//Check if the symbol string is an array, i.e. contains "[ ]"
FUNCTION F_CheckIsArraySymbol : BOOL
VAR_INPUT
    sSymbolName : STRING;
END_VAR
VAR
    iOpenBrackLocation : INT;
    iClosedBracketLocation : INT;
END_VAR

iOpenBrackLocation := FIND(sSymbolName, '[');
iClosedBracketLocation := FIND(sSymbolName, ']');

IF iOpenBrackLocation <> 0 AND iClosedBracketLocation > iOpenBrackLocation THEN
    F_CheckIsArraySymbol := TRUE;

ELSE
    F_CheckIsArraySymbol := FALSE;
END_IF

END_FUNCTION

(* stored: Version 1.1.0.1, ProductVersion 3.1.4024.12
   POU F_CheckIsArraySymbol: Id {fd4981a9-65d4-4598-983c-280485c47d3b}, SpecialFunc None *)
